// TwinCAT 3 PLC project DevelopmentProject
// ProgramVersion: 3.1.4024.0
// libraries:
//   Tc2_Standard, * (Beckhoff Automation GmbH)
//   Tc2_System, * (Beckhoff Automation GmbH)
//   Tc3_Module, * (Beckhoff Automation GmbH)
//   VisuSymbols,3.5.10.0,System
// project tree:
//   DUTs/ cylinder2IO.TcDUT, position_status.TcDUT, _2_position.TcDUT
//   / GlobalTextList.TcGTLO, PlcTask.TcTTO, Visualization Manager.TcVMO (not stored)
//   POUs/ Cylinder.TcPOU, TargetMAIN.TcPOU
//   VISUs/ Visualization.TcVIS
// real-time tasks:
//   TASK PlcTask: cycle T#10ms, priority 20, ADS port 350
//   TASK PlcTask1: cycle T#5ms, priority 21, ADS port 351
// I/O:
//   DEVICE Device 3 (EtherCAT), AmsNetId 10.200.64.8.4.1
//     Term 1 (EK1100) [EK1100 EtherCAT Coupler (2A E-Bus)]
//       Term 2 (EL1012) [EL1012 2Ch. Dig. Input 24V, 10µs]
//       Term 3 (EL2521) [EL2521 1Ch. Pulse Train Output]
//       Term 4 (EL2004) [EL2004 4Ch. Dig. Output 24V, 0.5A]
//       Term 5 (EL3152) [EL3152 2Ch. Ana Input 4-20mA]
//       Term 6 (EL9576) [EL9576 Brake chopper terminal]
//       Term 7 (EL4122) [EL4122 2Ch. Ana. Output  4-20mA, 16bit]
//       Term 8 (EL5101) [EL5101 1Ch. Inc. Encoder 5V]
//       Term 9 (EL6695) [EL6695 EtherCAT Bridge terminal (Primary)]
//       Term 10 (EK1122) [EK1122 2 port EtherCAT junction]
//       Term 11 (EL9011) [EL9011 End Terminal]
//   DEVICE Device 1 (EtherCAT Simulation), AmsNetId 10.200.64.8.2.1
//     Term 1 (EK1100) // EK1100-0000-0017
//     Term 2 (EL1012) // EL1012-0000-0016
//     Term 3 (EL2521) // EL2521-0000-1022
//     Term 4 (EL2004) // EL2004-0000-0016
//     Term 5 (EL3152) // EL3152-0000-0019
//     Term 6 (EL9576) // EL9576-0000-0021
//     Term 7 (EL4122) // EL4122-0000-1020
//     Term 8 (EL5101) // EL5101-0000-1024
//     Term 9 (EL6695) // EL6695-0000-0004
//     Term 10 (EK1122) // EK1122-0000-0017
// variable links:
//   DevelopmentProject/DevelopmentProject Instance <-> Device 3 (EtherCAT)/Term 1 (EK1100)/Term 2 (EL1012)
//     PlcTask Inputs/TargetMAIN.cylinder_1_io.pull_sensor <-> Channel 2/Input
//     PlcTask Inputs/TargetMAIN.cylinder_1_io.push_sensor <-> Channel 1/Input
//   DevelopmentProject/DevelopmentProject Instance <-> Device 3 (EtherCAT)/Term 1 (EK1100)/Term 4 (EL2004)
//     PlcTask Outputs/TargetMAIN.cylinder_1_io.pull_output <-> Channel 2/Output
//     PlcTask Outputs/TargetMAIN.cylinder_1_io.push_output <-> Channel 1/Output
//   SimulationProject/SimulationProject Instance <-> Device 1 (EtherCAT Simulation)/Term 2 (EL1012)
//     PlcTask Outputs/SimulationMAIN.io._pull_sensor <-> Channel 2/Input
//     PlcTask Outputs/SimulationMAIN.io._push_sensor <-> Channel 1/Input
//   SimulationProject/SimulationProject Instance <-> Device 1 (EtherCAT Simulation)/Term 4 (EL2004)
//     PlcTask Inputs/SimulationMAIN.io._pull_output <-> Channel 2/Output
//     PlcTask Inputs/SimulationMAIN.io._push_output <-> Channel 1/Output

CONFIGURATION DevelopmentProject
    RESOURCE PLC ON TwinCAT3
        TASK PlcTask(INTERVAL := T#10ms, PRIORITY := 20);
        PROGRAM TargetMAIN WITH PlcTask : TargetMAIN;
    END_RESOURCE
END_CONFIGURATION

// ---- DUTs/cylinder2IO.TcDUT
TYPE cylinder2IO :
STRUCT
	pull_sensor	AT%I*	:BOOL;
	push_sensor	AT%I*	:BOOL;
	pull_output AT%Q*	:BOOL;
	push_output AT%Q*	:BOOL;
END_STRUCT
END_TYPE

// ---- DUTs/position_status.TcDUT
{attribute 'qualified_only'}
{attribute 'strict'}
TYPE position_status :
(
	unknown := 0,
	inposition,
	moving
);
END_TYPE

// ---- DUTs/_2_position.TcDUT
{attribute 'qualified_only'}
{attribute 'strict'}
TYPE _2_position :
(
	position_1 := 0,
	position_2
);
END_TYPE

// ---- POUs/TargetMAIN.TcPOU
PROGRAM TargetMAIN
VAR
	cylinder_1 :Cylinder;
	cylinder_1_io :cylinder2IO;
	moving_overtime:	REAL := 5.0;
	push_stabilization: REAL := 500;
	pull_stabilization: REAL := 500;
	stroke_interval_time: REAL := 3.0;
	inposition : BOOL;
END_VAR


cylinder_1.limit_time := REAL_TO_TIME(moving_overtime * 1000);
cylinder_1.push_edge_time := REAL_TO_TIME(push_stabilization);
cylinder_1.pull_edge_time := REAL_TO_TIME(pull_stabilization);
cylinder_1.stroke_wait_time := REAL_TO_TIME(stroke_interval_time * 1000);

cylinder_1(io:=cylinder_1_io);

IF cylinder_1.status = position_status.inposition THEN
	inposition := TRUE;
ELSE
	inposition := FALSE;
END_IF

END_PROGRAM

// ---- POUs/Cylinder.TcPOU
FUNCTION_BLOCK Cylinder
VAR_INPUT
	bExecute: BOOL;
	command_activate: BOOL;
	push_edge_time: TIME := T#0.5S;
	pull_edge_time: TIME := T#0.5S;
	limit_time	: TIME := T#3S;
	keep_actuator : BOOL := FALSE;
	stroke_wait_time: TIME := T#5S;
END_VAR
VAR_OUTPUT
	status: position_status := position_status.unknown;
	position: _2_position;
	current_position: UINT;
	bError:BOOL;
END_VAR
VAR
	push_command: BOOL;
	pull_command: BOOL;
	edge_timer:Tc2_Standard.TON;
	limit_timer:Tc2_Standard.TON;
	stroke_wait_timer: Tc2_Standard.TON;
	last_cycle_position: _2_position;
	last_cycle_status : position_status;
END_VAR

VAR_IN_OUT
	io: cylinder2IO;
END_VAR

IF bExecute THEN
	stroke_wait_timer(IN := last_cycle_position = position, PT := stroke_wait_time);
	CASE position OF
		_2_position.position_2:
			IF stroke_wait_timer.Q THEN
				push_command := FALSE;
				pull_command := TRUE;				
			END_IF
		_2_position.position_1:
			IF stroke_wait_timer.Q THEN
				push_command := TRUE;
				pull_command := FALSE;
			END_IF
	END_CASE
ELSE
	push_command := FALSE;
	pull_command := FALSE;
END_IF
last_cycle_position := position;

command_activate := push_command OR pull_command;
CASE status OF
	position_status.unknown:
		IF last_cycle_status = position_status.inposition THEN
			bError := TRUE;
		END_IF
		io.push_output := FALSE;
		io.pull_output := FALSE;
		IF bError THEN
			bError := command_activate;
		ELSE
			IF push_command AND position = _2_position.position_1 THEN
				status := position_status.moving;
			END_IF
			IF pull_command AND position = _2_position.position_2 THEN
				status := position_status.moving;
			END_IF
		END_IF
	position_status.inposition:
		edge_timer.IN := FALSE;
		
		CASE position OF
			_2_position.position_1:
				IF push_command	THEN
					status := position_status.moving;
				END_IF
				IF io.push_sensor OR NOT io.pull_sensor THEN
					status := position_status.unknown;
				END_IF
			_2_position.position_2:
				IF pull_command	THEN
					status := position_status.moving;
				END_IF
				IF NOT io.push_sensor OR io.pull_sensor THEN
					status := position_status.unknown;
				END_IF
		END_CASE
		
		IF keep_actuator THEN
			io.push_output := (position = _2_position.position_2);
			io.pull_output := (position = _2_position.position_1);
		ELSE
			io.push_output := FALSE;
			io.pull_output := FALSE;
		END_IF
		
	position_status.moving:
		IF push_command THEN
			edge_timer.PT := push_edge_time;
			IF io.push_sensor AND NOT io.pull_sensor THEN
				edge_timer.IN := TRUE;
				IF edge_timer.Q THEN
					position := _2_position.position_2;
					status := position_status.inposition;
				END_IF
			ELSE
				edge_timer.IN := FALSE;
			END_IF
			io.push_output := TRUE;
			io.pull_output := FALSE;
		END_IF
		IF pull_command THEN
			edge_timer.PT := pull_edge_time;
			IF NOT io.push_sensor AND io.pull_sensor THEN
				edge_timer.IN := TRUE;
				IF edge_timer.Q THEN
					position := _2_position.position_1;
					status := position_status.inposition;
				END_IF
			ELSE
				edge_timer.IN := FALSE;
			END_IF
			io.push_output := FALSE;
			io.pull_output := TRUE;
		END_IF

END_CASE


limit_timer(IN:=command_activate AND (status <> position_status.inposition), PT:=limit_time);
IF limit_timer.Q THEN
	status := position_status.unknown;
	bError := TRUE;
END_IF

edge_timer();

last_cycle_status := status;

END_FUNCTION_BLOCK

// ---- GlobalTextList.TcGTLO
TEXTLIST GlobalTextList
  846 = '%0.01f'
  913 = '%0.1f'
  238 = '%0.2f'
  382 = '%10i'
  5 = '%1f'
  371 = '%1i'
  166 = '%1S'
  136 = '%3.2f'
  284 = '%3f'
  864 = '%3i'
  746 = '%S'
  540 = 'Active'
  35 = 'Alarm'
  523 = 'In position'
  262 = 'Interval'
  476 = 'Keep excitation'
  997 = 'ms'
  198 = 'Over time'
  189 = 'Pull confirm'
  878 = 'Pull stabilization'
  1 = 'Push stabilization'
  380 = 'Push stroke'
  359 = 'Push wait'
  545 = 's'
  406 = 'Sta'
  72 = 'Start'
END_TEXTLIST

// ---- VISUs/Visualization.TcVIS
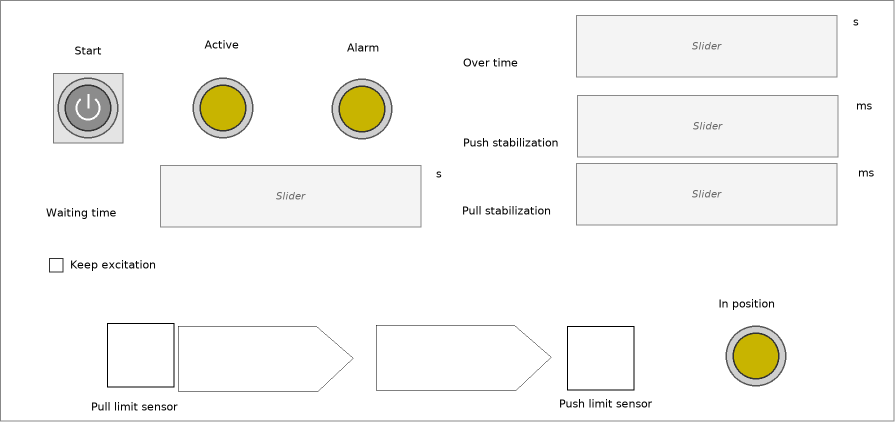
VISUALIZATION Visualization  // 895x422
    Lamp1 (188,73 70x70), variable: TargetMAIN.cylinder_1.bExecute, style: Lamp-Lamp1-Yellow
    PowerSwitch (53,73 70x70), variable: TargetMAIN.cylinder_1.bExecute, behaviour: TOGGLE, style: Switch-PowerSwitch-Gray
    Lamp1 (327,74 70x70), variable: TargetMAIN.cylinder_1.bError, style: Lamp-Lamp1-Yellow
    Slider (576,15 261x62), variable: TargetMAIN.moving_overtime, scale 0..10
    Label (460,48 150x30), "Over time"
    Slider (577,95 261x62), variable: TargetMAIN.push_stabilization, scale 0..1000
    Label (460,128 150x30), "Push stabilization"
    Label (459,196 150x30), "Pull stabilization"
    Slider (576,163 261x62), variable: TargetMAIN.pull_stabilization, scale 0..1000
    Label (43,198 150x30), "Waiting time"
    Slider (160,165 261x62), variable: TargetMAIN.stroke_interval_time, scale 0..10
    Label (288,33 150x30), "Alarm"
    Label (147,30 150x30), "Active"
    Label (13,36 150x30), "Start"
    Rectangle (107,323 67x64), colour toggle: TargetMAIN.cylinder_1_io.pull_sensor
    Rectangle (567,326 67x64), colour toggle: TargetMAIN.cylinder_1_io.push_sensor
    Label (853,91 40x30), "ms"
    Label (855,158 40x30), "ms"
    Label (850,7 40x30), "s"
    Label (433,159 40x30), "s"
    Checkbox (47,250 150x30), "Keep excitation", variable: TargetMAIN.cylinder_1.keep_actuator
    Polygon (376,325) (514,325) (551,357) (516,390) (376,390), colour toggle: TargetMAIN.cylinder_1.io.push_output
    Polygon (178,326) (316,326) (353,358) (318,391) (178,391), colour toggle: TargetMAIN.cylinder_1.io.pull_output
    Lamp1 (721,321 70x70), variable: TargetMAIN.inposition, style: Lamp-Lamp1-Yellow
    Label (672,289 150x30), "In position"
    Label (88,392 99x30), "Pull limit sensor"
    Label (556,389 99x30), "Push limit sensor"
END_VISUALIZATION
